// Mitsubishi GX Works2 project: dich_bit   PLC: FX3U/FX3UC

PROGRAM MAIN
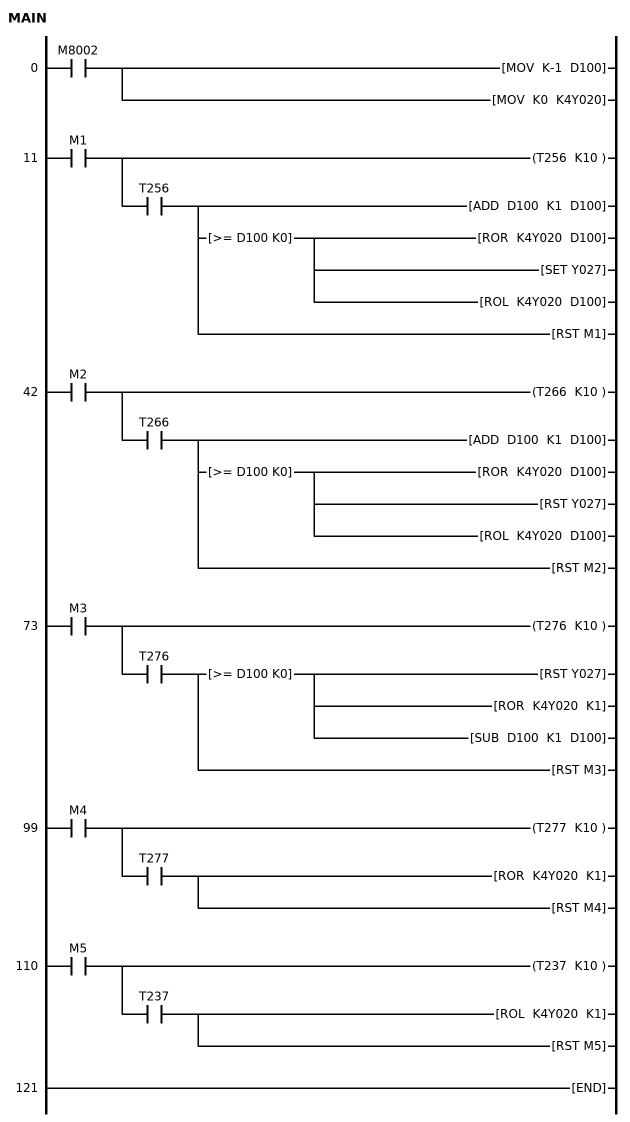
0     LD      M8002
      MOV     K-1 D100
      MOV     K0 K4Y020
11    LD      M1
      OUT     T256 K10
      AND     T256
      ADD     D100 K1 D100
      MPS
      AND>=   D100 K0
      ROR     K4Y020 D100
      SET     Y027
      ROL     K4Y020 D100
      MPP
      RST     M1
42    LD      M2
      OUT     T266 K10
      AND     T266
      ADD     D100 K1 D100
      MPS
      AND>=   D100 K0
      ROR     K4Y020 D100
      RST     Y027
      ROL     K4Y020 D100
      MPP
      RST     M2
73    LD      M3
      OUT     T276 K10
      AND     T276
      MPS
      AND>=   D100 K0
      RST     Y027
      ROR     K4Y020 K1
      SUB     D100 K1 D100
      MPP
      RST     M3
99    LD      M4
      OUT     T277 K10
      AND     T277
      ROR     K4Y020 K1
      RST     M4
110   LD      M5
      OUT     T237 K10
      AND     T237
      ROL     K4Y020 K1
      RST     M5
121   END
END_PROGRAM

// device comments not shown above
M0  ; add bit
